Omron CX-Programmer project NewProject (CX-Programmer 9.54)

# PLC NewPLC1: CP1E N30

## Global symbols (name address type ; comment)
0.00 BOOL  ; START_1
0.01 BOOL  ; RESET
0.02 BOOL  ; EMG
0.03 BOOL  ; A_MIN
0.04 BOOL  ; A_PLUS
0.05 BOOL  ; B_MIN
0.06 BOOL  ; B_PLUS
0.07 BOOL  ; C_MIN
0.08 BOOL  ; C_PLUS
0.09 BOOL  ; OBJ_SENS
0.10 BOOL  ; START_2
0.11 BOOL  ; SENS_OBJ
10.00 BOOL  ; TRIGGER_START
10.01 BOOL  ; INIT_POS
10.02 BOOL  ; STEP_1
10.03 BOOL  ; STEP_2
10.04 BOOL  ; STEP_3
10.05 BOOL  ; STEP_4
10.06 BOOL  ; STEP_5
10.07 BOOL  ; STEP_6
10.08 BOOL  ; END_STEP
10.09 BOOL  ; TRIG_RESET
10.10 BOOL  ; STEP_RST_1
10.11 BOOL  ; STEP_RST_2
10.12 BOOL  ; STEP_RST_3
10.13 BOOL  ; STEP_RST_END

## Program NewProgram1 (cyclic task 0)
Local symbols
START_2 BOOL

### Section Section1

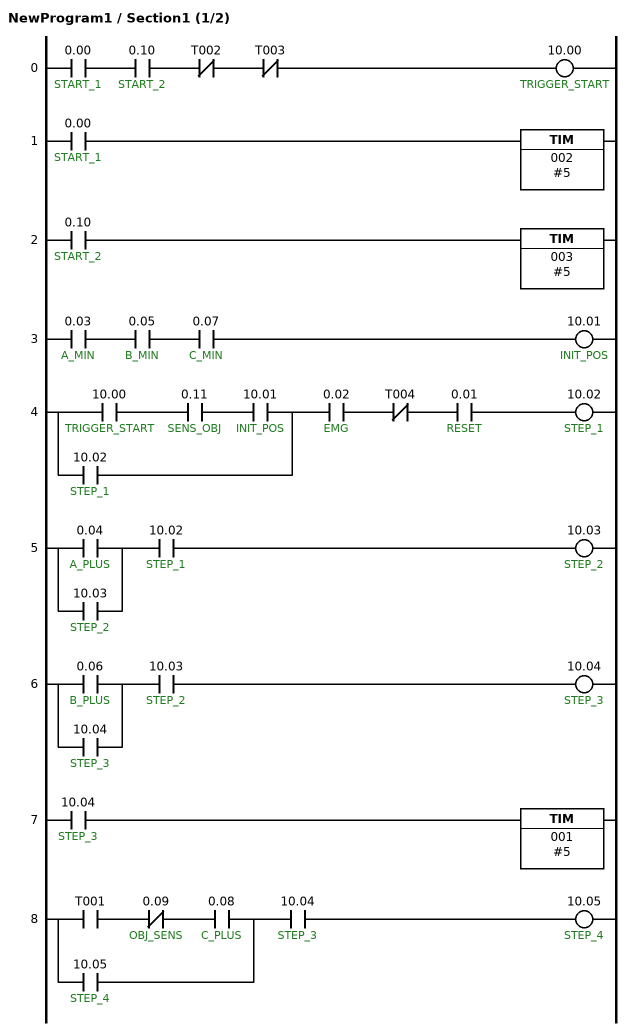
; rung 0
LD 0.00  ; START_1
AND 0.10  ; START_2
ANDNOT T002
ANDNOT T003
OUT 10.00  ; TRIGGER_START
; rung 1
LD 0.00  ; START_1
TIM 002 #5
; rung 2
LD 0.10  ; START_2
TIM 003 #5
; rung 3
LD 0.03  ; A_MIN
AND 0.05  ; B_MIN
AND 0.07  ; C_MIN
OUT 10.01  ; INIT_POS
; rung 4
LD 10.00  ; TRIGGER_START
AND 0.11  ; SENS_OBJ
AND 10.01  ; INIT_POS
OR 10.02  ; STEP_1
AND 0.02  ; EMG
ANDNOT T004
AND 0.01  ; RESET
OUT 10.02  ; STEP_1
; rung 5
LD 0.04  ; A_PLUS
OR 10.03  ; STEP_2
AND 10.02  ; STEP_1
OUT 10.03  ; STEP_2
; rung 6
LD 0.06  ; B_PLUS
OR 10.04  ; STEP_3
AND 10.03  ; STEP_2
OUT 10.04  ; STEP_3
; rung 7
LD 10.04  ; STEP_3
TIM 001 #5
; rung 8
LD T001
ANDNOT 0.09  ; OBJ_SENS
AND 0.08  ; C_PLUS
OR 10.05  ; STEP_4
AND 10.04  ; STEP_3
OUT 10.05  ; STEP_4

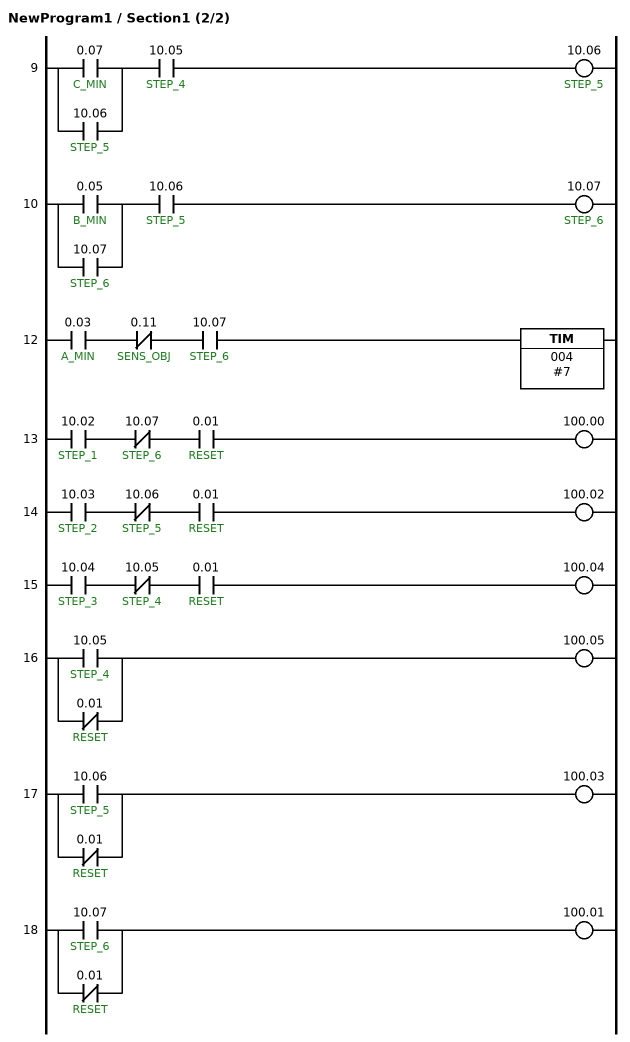
; rung 9
LD 0.07  ; C_MIN
OR 10.06  ; STEP_5
AND 10.05  ; STEP_4
OUT 10.06  ; STEP_5
; rung 10
LD 0.05  ; B_MIN
OR 10.07  ; STEP_6
AND 10.06  ; STEP_5
OUT 10.07  ; STEP_6
; rung 12
LD 0.03  ; A_MIN
ANDNOT 0.11  ; SENS_OBJ
AND 10.07  ; STEP_6
TIM 004 #7
; rung 13
LD 10.02  ; STEP_1
ANDNOT 10.07  ; STEP_6
AND 0.01  ; RESET
OUT 100.00
; rung 14
LD 10.03  ; STEP_2
ANDNOT 10.06  ; STEP_5
AND 0.01  ; RESET
OUT 100.02
; rung 15
LD 10.04  ; STEP_3
ANDNOT 10.05  ; STEP_4
AND 0.01  ; RESET
OUT 100.04
; rung 16
LD 10.05  ; STEP_4
ORNOT 0.01  ; RESET
OUT 100.05
; rung 17
LD 10.06  ; STEP_5
ORNOT 0.01  ; RESET
OUT 100.03
; rung 18
LD 10.07  ; STEP_6
ORNOT 0.01  ; RESET
OUT 100.01

### Section END
; rung 0
END(001)